FUNCTION F_ToAnyType : ST_AnyType
VAR_INPUT
    anyArg	: ANY;
END_VAR

F_ToAnyType.pValue := anyArg.pValue;
F_ToAnyType.nSize := anyArg.diSize;
F_ToAnyType.TypeClass := anyArg.TypeClass;

END_FUNCTION

(* stored: Version 1.1.0.1
   POU F_ToAnyType: Id {dadf5a57-eeb7-4a05-afb8-69b1ccd3a266}, SpecialFunc None *)
